# EPICS substitutions: apps/jscalerApp/Db/jscalers_wf_S3.substitutions
file "db/jscalers_wf_averages-1type-1sector.db" {
pattern { T S }
{ FADC 3 }
{ TRG 3 }
{ TDC 3 }
}
